{attribute 'qualified_only'}
TYPE E_ATM_States :
(
    Unknown := 0,
    OUT := 1,
    TARGET1 := 2,
    TARGET2 := 3,
    TARGET3 := 4,
    TARGET4 := 5,
    TARGET5 := 6,
    TARGET6 := 7,
    TARGET7 := 8
) UINT;
END_TYPE

(* stored: Version 1.1.0.1
   DUT E_ATM_States: Id {39e72780-ebe1-47a1-93c3-70f8a4ded457} *)
